Staubli VAL3: runHigh.pgx

public program runHigh()
begin
  call taskPartMade()
  call IMMTiming()
   call BtRobotOff()

  call secuTask1()
  call secuTask2()
end
